{attribute addProperty BoxType "AMP8000-0030-0103-0103"}
{attribute addProperty Id "Safe_Logic_StateUSINT811Cycle_CounterUSINT812"}
{attribute addProperty CRC "1874648931"}
{attribute addProperty SizeInBites "16"}
{attribute addProperty SizeInBytes "2"}
TYPE FSOE_6FBCDF63 :
STRUCT
	{attribute addProperty Name "Safe_Logic_State"}
	Safe_Logic_State : USINT;
	{attribute addProperty Name "Cycle_Counter"}
	Cycle_Counter : USINT;
END_STRUCT
END_TYPE

(* stored: Version 1.2.0.0, ProductVersion 3.1.4024.9
   DUT FSOE_6FBCDF63: Id {7d765bb6-60c0-43fb-8876-b4707234a0bc} *)
